{attribute 'qualified_only'}
{attribute 'strict'}
{attribute 'to_string'}
TYPE E_MoveMode  :
(
    DISCRETE_JOG:=0,
    DISCRETE_VELOCITY:=1,
    DISCRETE_RELATIVE:=2,
    DISCRETE_ABSOLUTE:=3,
    DISCRETE_MODULO:=4,
    DISCRETE_HOMING:=10
)INT;
END_TYPE

(* stored: Version 1.1.0.1
   DUT E_MoveMode: Id {84e949ba-0c00-4cd0-8823-2572cfa98b29} *)
